Staubli VAL3: buildList.pgx

program buildList()
  local bool l_bFound
  local num i
  local num l_nCount
  local num l_nSize
  local string l_sEvent
  local string l_sEmpty
begin
  // INIT the list
  l_sEmpty=""
  call use:stringCopy(l_sEmpty,sList)
  // filter the result??
  call prog:getSize(l_nSize)
  for i=0 to l_nSize-1
    call prog:get(l_sEvent,i)
    // patch for the #program
    if l_sEvent!=""
      //
      // use the filter ?
      //
      l_bFound=true
      if saveData:sProgFilter!=""
        l_bFound=find(l_sEvent,saveData:sProgFilter)!=-1
      endIf
      // add
      if l_bFound
        if (left(l_sEvent,1)=="#" and nProgID==2)
          call listAdd(l_sEvent)
        elseIf nProgID!=2 and left(l_sEvent,1)!="#" and l_sEvent!="HOME1" and l_sEvent!="HOME2"
          call listAdd(l_sEvent)
        endIf
        l_nCount=l_nCount+1
      endIf
    endIf
  endFor
end
